DATA_BLOCK "IN"
{ S7_Optimized_Access := 'FALSE' }
VERSION : 0.1
NON_RETAIN
   STRUCT
      "1层上行呼梯按钮" : Bool;
      "2层上行呼梯按钮" : Bool;
      "3层上行呼梯按钮" : Bool;
      "4层上行呼梯按钮" : Bool;
      "5层上行呼梯按钮" : Bool;
      "6层上行呼梯按钮" : Bool;
      "7层上行呼梯按钮" : Bool;
      "8层上行呼梯按钮" : Bool;
      "9层上行呼梯按钮" : Bool;
      "2层下行呼梯按钮" : Bool;
      "3层下行呼梯按钮" : Bool;
      "4层下行呼梯按钮" : Bool;
      "5层下行呼梯按钮" : Bool;
      "6层下行呼梯按钮" : Bool;
      "7层下行呼梯按钮" : Bool;
      "8层下行呼梯按钮" : Bool;
      "9层下行呼梯按钮" : Bool;
      "10层下行呼梯按钮" : Bool;
      "1号梯轿内选层按钮1" : Bool;
      "1号梯轿内选层按钮2" : Bool;
      "1号梯轿内选层按钮3" : Bool;
      "1号梯轿内选层按钮4" : Bool;
      "1号梯轿内选层按钮5" : Bool;
      "1号梯轿内选层按钮6" : Bool;
      "1号梯轿内选层按钮7" : Bool;
      "1号梯轿内选层按钮8" : Bool;
      "1号梯轿内选层按钮9" : Bool;
      "1号梯轿内选层按钮10" : Bool;
      "1号梯轿内开门按钮" : Bool;
      "1号梯轿内关门按钮" : Bool;
      "1号梯光幕信号" : Bool;
      "1号梯检修信号" : Bool;
      "1号梯轿厢门锁信号" : Bool;
      "1号梯1楼层门锁信号" : Bool;
      "1号梯2楼层门锁信号" : Bool;
      "1号梯3楼层门锁信号" : Bool;
      "1号梯4楼层门锁信号" : Bool;
      "1号梯5楼层门锁信号" : Bool;
      "1号梯6楼层门锁信号" : Bool;
      "1号梯7楼层门锁信号" : Bool;
      "1号梯8楼层门锁信号" : Bool;
      "1号梯9楼层门锁信号" : Bool;
      "1号梯10楼层门锁信号" : Bool;
      "1号梯开门到位" : Bool;
      "1号梯关门到位" : Bool;
      "1号梯上平层信号" : Bool;
      "1号梯下平层信号" : Bool;
      "1号梯上端站第1限位" : Bool;
      "1号梯上端站第2限位" : Bool;
      "1号梯下端站第1限位" : Bool;
      "1号梯下端站第2限位" : Bool;
      "2号梯轿内选层按钮1" : Bool;
      "2号梯轿内选层按钮2" : Bool;
      "2号梯轿内选层按钮3" : Bool;
      "2号梯轿内选层按钮4" : Bool;
      "2号梯轿内选层按钮5" : Bool;
      "2号梯轿内选层按钮6" : Bool;
      "2号梯轿内选层按钮7" : Bool;
      "2号梯轿内选层按钮8" : Bool;
      "2号梯轿内选层按钮9" : Bool;
      "2号梯轿内选层按钮10" : Bool;
      "2号梯轿内开门按钮" : Bool;
      "2号梯轿内关门按钮" : Bool;
      "2号梯光幕信号" : Bool;
      "2号梯检修信号" : Bool;
      "2号梯轿厢门锁信号" : Bool;
      "2号梯1楼层门锁信号" : Bool;
      "2号梯2楼层门锁信号" : Bool;
      "2号梯3楼层门锁信号" : Bool;
      "2号梯4楼层门锁信号" : Bool;
      "2号梯5楼层门锁信号" : Bool;
      "2号梯6楼层门锁信号" : Bool;
      "2号梯7楼层门锁信号" : Bool;
      "2号梯8楼层门锁信号" : Bool;
      "2号梯9楼层门锁信号" : Bool;
      "2号梯10楼层门锁信号" : Bool;
      "2号梯开门到位" : Bool;
      "2号梯关门到位" : Bool;
      "2号梯上平层信号" : Bool;
      "2号梯下平层信号" : Bool;
      "2号梯上端站第1限位" : Bool;
      "2号梯上端站第2限位" : Bool;
      "2号梯下端站第1限位" : Bool;
      "2号梯下端站第2限位" : Bool;
      "3号梯轿内选层按钮1" : Bool;
      "3号梯轿内选层按钮2" : Bool;
      "3号梯轿内选层按钮3" : Bool;
      "3号梯轿内选层按钮4" : Bool;
      "3号梯轿内选层按钮5" : Bool;
      "3号梯轿内选层按钮6" : Bool;
      "3号梯轿内选层按钮7" : Bool;
      "3号梯轿内选层按钮8" : Bool;
      "3号梯轿内选层按钮9" : Bool;
      "3号梯轿内选层按钮10" : Bool;
      "3号梯轿内开门按钮" : Bool;
      "3号梯轿内关门按钮" : Bool;
      "3号梯光幕信号" : Bool;
      "3号梯检修信号" : Bool;
      "3号梯轿厢门锁信号" : Bool;
      "3号梯1楼层门锁信号" : Bool;
      "3号梯2楼层门锁信号" : Bool;
      "3号梯3楼层门锁信号" : Bool;
      "3号梯4楼层门锁信号" : Bool;
      "3号梯5楼层门锁信号" : Bool;
      "3号梯6楼层门锁信号" : Bool;
      "3号梯7楼层门锁信号" : Bool;
      "3号梯8楼层门锁信号" : Bool;
      "3号梯9楼层门锁信号" : Bool;
      "3号梯10楼层门锁信号" : Bool;
      "3号梯开门到位" : Bool;
      "3号梯关门到位" : Bool;
      "3号梯上平层信号" : Bool;
      "3号梯下平层信号" : Bool;
      "3号梯上端站第1限位" : Bool;
      "3号梯上端站第2限位" : Bool;
      "3号梯下端站第1限位" : Bool;
      "3号梯下端站第2限位" : Bool;
      自动运行信号 : Bool;
      "1号梯当前载重量" : Word;
      "2号梯当前载重量" : Word;
      "3号梯当前载重量" : Word;
   END_STRUCT;


BEGIN

END_DATA_BLOCK

